TYPE ST_PositionXY :
STRUCT
  X : REAL;
  Y : REAL;
END_STRUCT
END_TYPE

(* stored: Version 1.1.0.1, ProductVersion 3.1.4024.12
   DUT ST_PositionXY: Id {99799802-56bd-4dfb-8f26-d861a8b2a5fe} *)
